PROGRAM Analog_PRG
VAR
	

AI_Input : INT;
AO_Output : INT;
AO_Unscrambler : INT;
AO_Grading : INT;
AO_SawFeedChain: INT;

// --- Analog routing logic ---
// Selection = 1..3 (from HMI dropdown)
Selection : ARRAY[1..3] OF BOOL;  // 1=Unscrambler, 2=Grading, 3=SawFeed



END_VAR

//---------------------------Defaults-----------------------------
AO_Unscrambler := 0;
AO_Grading := 0;
AO_SawFeedChain := 0;



AI_INT := AI_Input;

UnscramblerVFD1speed := AO_Unscrambler;
GradingVFD2speed := AO_Grading;
SawFeedVFD3speed := AO_SawFeedChain;







CASE Selection OF
//Selection 1 - Unscrambler	
1:  

AO_Unscrambler := AI_Input;
AO_Grading := 0;
AO_SawFeedChain := 0;

// Selection 2 - Grading
2:  

AO_Grading := AI_Input;
AO_Unscrambler := 0;
AO_SawFeedChain := 0;


// Selection 3 - Saw FeedChain
3:  

AO_SawFeedChain := AI_Input;
AO_Unscrambler := 0;
AO_Grading := 0;

// --- Default (nothing selected) ---
ELSE
    AO_Unscrambler := 0;
    AO_Grading := 0;
    AO_SawFeedChain := 0;

END_CASE

END_PROGRAM

(* stored: Version 1.1.0.1
   POU Analog_PRG: Id {52760586-22c0-4906-a346-d41bff646391}, SpecialFunc None *)
